// TwinCAT 3 PLC project Untitled1
// ProgramVersion: 3.1.4023.0
// libraries:
//   Tc2_Standard, * (Beckhoff Automation GmbH)
//   Tc2_System, * (Beckhoff Automation GmbH)
//   Tc3_Module, * (Beckhoff Automation GmbH)
// project tree:
//   / PlcTask.TcTTO
//   POUs/ MAIN.TcPOU, TONReset.TcPOU
// real-time tasks:
//   TASK PlcTask: cycle T#10ms, priority 20, ADS port 350
// motion (NC):
//   TASK NC-Task 1 SAF: cycle T#2ms, priority 4, ADS port 501
//   TASK NC-Task 1 SVB: cycle T#10ms, priority 8, ADS port 511
//   AXIS Axis 1 (id 1)
//     OtherSettings: AllowMotionCmdToSlave=true
//     encoder EncType=19
//       EncPara: MaxCount=#xffffffff
//     drive DrvType=16
//       DrvPara: MaxCount=#xffffffff
//         Analog: TorqueSetpointScale=10, ScaleFactorActTorque=0.1
//         TimeComp: TaskDelayCycles=1
//     controller CtrType=1
//       CtrPara: PriorControlFactor=1
//         Observer: BandWidth=20
//   AXIS Axis 2 (id 2)
//     OtherSettings: AllowMotionCmdToSlave=true
//     encoder EncType=19
//       EncPara: MaxCount=#xffffffff
//     drive DrvType=16
//       DrvPara: MaxCount=#xffffffff
//         Analog: TorqueSetpointScale=10, ScaleFactorActTorque=0.1
//         TimeComp: TaskDelayCycles=1
//     controller CtrType=1
//       CtrPara: PriorControlFactor=1
//         Observer: BandWidth=20
// I/O:
//   DEVICE Device 1 (EtherCAT), AmsNetId 192.168.4.11.2.1
//     Term 11 (EK1914) [EK1914, 2 Ch. Safety Input/Output 24V,  TwinSAFE]
//       modules: Module 1 (FSOE), Module 2 (DIO)
//       Term 12 (EL9410) [EL9410 E-Bus Power Supplier  (Diagnostics)]
//       Term 13 (EL3164) [EL3164 4Ch. Ana. Input 0-10V]
//       Term 14 (EL4104) [EL4104 4Ch. Ana. Output 0-10V, 16bit]
//       Term 15 (EL6614) [EL6614 4 Port Switch (Ethernet, CoE)]
//       Term 16 (EL6002) [EL6002 Interface 2Ch. (RS232)]
//       Term 17 (EL9410) [EL9410 E-Bus Power Supplier  (Diagnostics)]
//       Term 18 (EL7201-9014) [EL7201-9014 1Ch. MDP742 Servo motor output stage with OCT (50V, 2.8A RMS) and STO input]
//       Term 19 (EL7201-9014) [EL7201-9014 1Ch. MDP742 Servo motor output stage with OCT (50V, 2.8A RMS) and STO input]
//       Term 20 (EL9011) [EL9011 End Terminal]
// variable links:
//   Untitled1/Untitled1 Instance <-> Device 1 (EtherCAT)/Term 11 (EK1914)
//     PlcTask Inputs/MAIN.xSigC <-> Module 2 (DIO)/DIO Inputs/Input 0
//     PlcTask Inputs/MAIN.xSigO <-> Module 2 (DIO)/DIO Inputs/Input 1
//   Untitled1/Untitled1 Instance <-> Device 1 (EtherCAT)/Term 11 (EK1914)/Term 13 (EL3164)
//     PlcTask Inputs/MAIN.iHumidityRaw <-> AI Standard Channel 1/Value
//     PlcTask Inputs/MAIN.iTempRaw <-> AI Standard Channel 2/Value

CONFIGURATION Untitled1
    RESOURCE PLC ON TwinCAT3
        TASK PlcTask(INTERVAL := T#10ms, PRIORITY := 20);
        PROGRAM MAIN WITH PlcTask : MAIN;
    END_RESOURCE
END_CONFIGURATION

// ---- POUs/MAIN.TcPOU
PROGRAM MAIN
VAR
	xBool	: BOOL;
	xSigC	AT %I* : BOOL;
	xSigO	AT %I* : BOOL;
	iHumidityRaw AT %I* : INT;
	iTempRaw	AT %I* : INT;
	fbTONR	: TONReset;
END_VAR

fbTONR(PT	:= T#4S);

IF fbTONR.rtTimerDone.Q THEN
	xBool	:= TRUE;
END_IF

END_PROGRAM

// ---- POUs/TONReset.TcPOU
FUNCTION_BLOCK TONReset EXTENDS TON
VAR_INPUT
END_VAR
VAR_OUTPUT
	rtTimerDone	: R_TRIG;
END_VAR
VAR
END_VAR

SUPER^();

rtTimerDone(CLK	:= THIS^.Q);

IF THIS^.Q THEN 
	THIS^.IN	:= FALSE;
END_IF

END_FUNCTION_BLOCK
